TYPE ST_ElementBase :
(**************************************************************************************
 * 	Application		:	BoxControl Framework
 *	Revision		:	$Revision: 404529 $
 *	Revision date	:	$Date: 2018-04-23 08:21:38 +0200 (Mo., 23 Apr 2018) $
 *	Last changed by	:	$Author: b7bolm $
 *	URL				:	$URL: http://almscdc.swisslog.com/repo/SWPD/Development/BoxControlFramework/20_Release/trunk/01_Software/BCF/BCF/JumpStart/20_Product/10_App/13_Elements/10_Lib/10_Conv/01_DUTs/ST_ElementBase.TcDUT $
 *
 *	Purpose			:	Basis element data
 *
 * ------------------------------------------------------------------------------------
 *	Copyright Swisslog [IP AG], Switzerland. All rights reserved.
 * 
 * ------------------------------------------------------------------------------------
 *	
 * 	Revision History: 
 *
 * 	VERSION			DATE			INITIALS			DESCRIPTION
 *	0.1				01.01.2001		swl					Example
 *
 **************************************************************************************)
STRUCT
	eMsgType				: E_ITC_MsgTypeConv; // ITC message
	eReturnCode				: E_ErrorConv; // Error code
	FunctionStopped			: BOOL; // Function are stopped
	Idx						: INT; // Iterator
	MemberState				: ST_PositionState; // Member state
	FunctionOrdersEmpty		: ST_FunctionOrders;
	OperationStateEmpty		: ST_PositionState;
	ESQ						: ST_ITC_ESQ; // ITC message
	ECQ						: ST_ITC_ECQ; // ITC message
	MCQ						: ST_ITC_MCQ; // ITC message	
END_STRUCT
END_TYPE

(* stored: Version 1.1.0.1, ProductVersion 3.1.4022.12
   DUT ST_ElementBase: Id {1b8784c4-2d26-4a4e-b5c5-554e0fbc7511} *)
